PROGRAM C21_CamerasCtrl
VAR
END_VAR

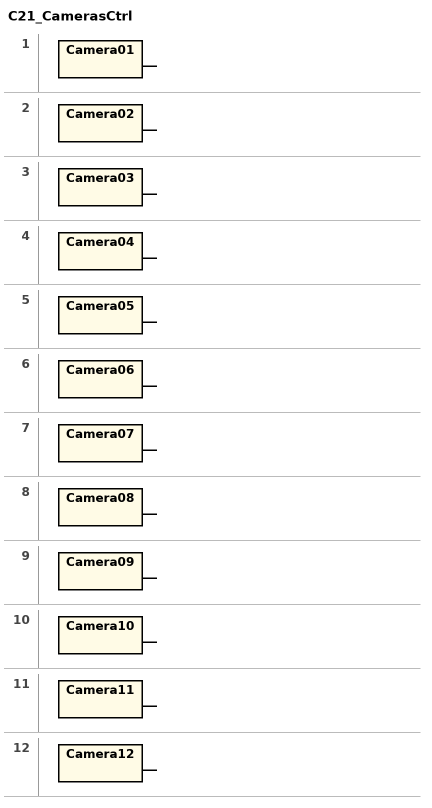
// NETWORK 1
Camera01();

// NETWORK 2
Camera02();

// NETWORK 3
Camera03();

// NETWORK 4
Camera04();

// NETWORK 5
Camera05();

// NETWORK 6
Camera06();

// NETWORK 7
Camera07();

// NETWORK 8
Camera08();

// NETWORK 9
Camera09();

// NETWORK 10
Camera10();

// NETWORK 11
Camera11();

// NETWORK 12
Camera12();

ACTION Camera01:
(*********************************************************CAMERA 01**********************************************************************)

(*stMasterListCameraOptions		: ST_SCANNER_Options := (eScannerType := E_MV_420_FULL, nImageBuffer := 1, nExpectedResp := 1);*)
IF gProcess.ePackAggregationMode <> E_SYSTEM_PAOL_2CAM AND gProcess.ePackAggregationMode <> E_SYSTEM_PAOL_3CAM  THEN

	gDevice.aCameraLightingIntensity[1] := F_SCANNER_LightingIntensity(gDevice.stMachineConfig.aCameraSettings[1].nLightingIntensity);

	gDevice.aCameraControl[1].stOptions.bUseExternalLight := gDevice.stMachineConfig.aCameraSettings[1].bUseExternalLight;
	gDevice.aCameraControl[1].stOptions.eScannerType	:= gDevice.stMachineConfig.aCameraSettings[1].eScannerType;

	IF gDevice.aCameraControl[1].stOptions.eScannerType = E_SCANNER_DeviceType.V430F THEN

		gDevice.aCameraControl[1].stOptions.nImageBuffer	:= 1;
		gDevice.aCameraControl[1].stOptions.nExpectedResp := 1;
		gDevice.aCameraControl[1].nReqProgram := 1;

	ELSE

		gDevice.aCameraControl[1].stOptions.nImageBuffer 	:= gDevice.stMachineConfig.aCameraSettings[1].nImageBuffer;
		gDevice.aCameraControl[1].stOptions.nExpectedResp := gDevice.stMachineConfig.aCameraSettings[1].nExpectedResp;

		CASE gDevice.stMachineConfig.aCameraSettings[1].eExpectedType OF
				E_SCANNER_CodeType.DATAMARTIX:
					gDevice.aCameraControl[1].nReqProgram := 1;
				E_SCANNER_CodeType.DOTCODE:
					gDevice.aCameraControl[1].nReqProgram := 2;
				E_SCANNER_CodeType.QR:
					gDevice.aCameraControl[1].nReqProgram := 3;
				E_SCANNER_CodeType.CODE128:
					gDevice.aCameraControl[1].nReqProgram := 4;
			ELSE
				gDevice.aCameraControl[1].nReqProgram := 1;
			END_CASE
	END_IF
END_IF
END_ACTION

ACTION Camera02:
(*********************************************************CAMERA 02**********************************************************************)
(*stPackAggregationCameraOptions		: ST_SCANNER_Options := (eScannerType := E_MV_420_FULL, nImageBuffer := 1, nExpectedResp := 1);*)
(*stPackAggregationCameraOptions		: ST_SCANNER_Options := (eScannerType := E_MV_None, nImageBuffer := 1, nExpectedResp := 5);*)
(*stPackAggregationCameraOptions		: ST_SCANNER_Options := (eScannerType := E_MV_None, nImageBuffer := 1, nExpectedResp := 2);*)
IF gProcess.ePackAggregationMode <> E_SYSTEM_PAOL_2CAM AND gProcess.ePackAggregationMode <> E_SYSTEM_PAOL_3CAM  THEN

	gDevice.aCameraLightingIntensity[2] := F_SCANNER_LightingIntensity(gDevice.stMachineConfig.aCameraSettings[2].nLightingIntensity);

	gDevice.aCameraControl[2].stOptions.bUseExternalLight := gDevice.stMachineConfig.aCameraSettings[2].bUseExternalLight;
	gDevice.aCameraControl[2].stOptions.eScannerType	:= gDevice.stMachineConfig.aCameraSettings[2].eScannerType;

	IF gDevice.aCameraControl[2].stOptions.eScannerType = E_SCANNER_DeviceType.V430F THEN

		gDevice.aCameraControl[2].stOptions.nImageBuffer	:= 1;
		gDevice.aCameraControl[2].stOptions.nExpectedResp := 1;
		gDevice.aCameraControl[2].nReqProgram := 1;

	ELSE

		gDevice.aCameraControl[2].stOptions.nImageBuffer 	:= gDevice.stMachineConfig.aCameraSettings[2].nImageBuffer;
		gDevice.aCameraControl[2].stOptions.nExpectedResp := gDevice.stMachineConfig.aCameraSettings[2].nExpectedResp;

		CASE gDevice.stMachineConfig.aCameraSettings[2].eExpectedType OF
				E_SCANNER_CodeType.DATAMARTIX:
					gDevice.aCameraControl[2].nReqProgram := 1;
				E_SCANNER_CodeType.DOTCODE:
					gDevice.aCameraControl[2].nReqProgram := 2;
				E_SCANNER_CodeType.QR:
					gDevice.aCameraControl[2].nReqProgram := 3;
				E_SCANNER_CodeType.CODE128:
					gDevice.aCameraControl[2].nReqProgram := 4;
			ELSE
				gDevice.aCameraControl[2].nReqProgram := 1;
			END_CASE
	END_IF
END_IF
END_ACTION

ACTION Camera03:
(*********************************************************CAMERA 03**********************************************************************)

(*stPackAggregationCameraOptions		: ST_SCANNER_Options := (eScannerType := E_MV_420_FULL, nImageBuffer := 1, nExpectedResp := 1);*)
(*stPackAggregationCameraOptions		: ST_SCANNER_Options := (eScannerType := E_MV_None, nImageBuffer := 1, nExpectedResp := 5);*)
(*stPackAggregationCameraOptions		: ST_SCANNER_Options := (eScannerType := E_MV_None, nImageBuffer := 1, nExpectedResp := 2);*)
IF gProcess.ePackAggregationMode <> E_SYSTEM_PAOL_2CAM AND gProcess.ePackAggregationMode <> E_SYSTEM_PAOL_3CAM  THEN

	gDevice.aCameraLightingIntensity[3] := F_SCANNER_LightingIntensity(gDevice.stMachineConfig.aCameraSettings[3].nLightingIntensity);

	gDevice.aCameraControl[3].stOptions.bUseExternalLight := gDevice.stMachineConfig.aCameraSettings[3].bUseExternalLight;
	gDevice.aCameraControl[3].stOptions.eScannerType	:= gDevice.stMachineConfig.aCameraSettings[3].eScannerType;

	IF gDevice.aCameraControl[3].stOptions.eScannerType = E_SCANNER_DeviceType.V430F THEN

		gDevice.aCameraControl[3].stOptions.nImageBuffer	:= 1;
		gDevice.aCameraControl[3].stOptions.nExpectedResp := 1;
		gDevice.aCameraControl[3].nReqProgram := 1;

	ELSE

		gDevice.aCameraControl[3].stOptions.nImageBuffer 	:= gDevice.stMachineConfig.aCameraSettings[3].nImageBuffer;
		gDevice.aCameraControl[3].stOptions.nExpectedResp := gDevice.stMachineConfig.aCameraSettings[3].nExpectedResp;

		CASE gDevice.stMachineConfig.aCameraSettings[3].eExpectedType OF
				E_SCANNER_CodeType.DATAMARTIX:
					gDevice.aCameraControl[3].nReqProgram := 1;
				E_SCANNER_CodeType.DOTCODE:
					gDevice.aCameraControl[3].nReqProgram := 2;
				E_SCANNER_CodeType.QR:
					gDevice.aCameraControl[3].nReqProgram := 3;
				E_SCANNER_CodeType.CODE128:
					gDevice.aCameraControl[3].nReqProgram := 4;
			ELSE
				gDevice.aCameraControl[3].nReqProgram := 1;
			END_CASE
	END_IF
END_IF
END_ACTION

ACTION Camera04:
(*********************************************************CAMERA 04**********************************************************************)
gDevice.aCameraLightingIntensity[4] := F_SCANNER_LightingIntensity(gDevice.stMachineConfig.aCameraSettings[4].nLightingIntensity);

gDevice.aCameraControl[4].stOptions.bUseExternalLight := gDevice.stMachineConfig.aCameraSettings[4].bUseExternalLight;
gDevice.aCameraControl[4].stOptions.eScannerType	:= gDevice.stMachineConfig.aCameraSettings[4].eScannerType;

IF gDevice.aCameraControl[4].stOptions.eScannerType = E_SCANNER_DeviceType.V430F THEN

	gDevice.aCameraControl[4].stOptions.nImageBuffer	:= 1;
	gDevice.aCameraControl[4].stOptions.nExpectedResp := 1;
	gDevice.aCameraControl[4].nReqProgram := 1;

ELSE

	gDevice.aCameraControl[4].stOptions.nImageBuffer 	:= gDevice.stMachineConfig.aCameraSettings[4].nImageBuffer;
	gDevice.aCameraControl[4].stOptions.nExpectedResp := gDevice.stMachineConfig.aCameraSettings[4].nExpectedResp;

	CASE gDevice.stMachineConfig.aCameraSettings[4].eExpectedType OF
			E_SCANNER_CodeType.DATAMARTIX:
				gDevice.aCameraControl[4].nReqProgram := 1;
			E_SCANNER_CodeType.DOTCODE:
				gDevice.aCameraControl[4].nReqProgram := 2;
			E_SCANNER_CodeType.QR:
				gDevice.aCameraControl[4].nReqProgram := 3;
			E_SCANNER_CodeType.CODE128:
				gDevice.aCameraControl[4].nReqProgram := 4;
		ELSE
			gDevice.aCameraControl[4].nReqProgram := 1;
		END_CASE
END_IF
END_ACTION

ACTION Camera05:
(*********************************************************CAMERA 05**********************************************************************)
gDevice.aCameraLightingIntensity[5] := F_SCANNER_LightingIntensity(gDevice.stMachineConfig.aCameraSettings[5].nLightingIntensity);

gDevice.aCameraControl[5].stOptions.bUseExternalLight := gDevice.stMachineConfig.aCameraSettings[5].bUseExternalLight;
gDevice.aCameraControl[5].stOptions.eScannerType	:= gDevice.stMachineConfig.aCameraSettings[5].eScannerType;
gDevice.aCameraControl[5].stOptions.nImageBuffer 	:= gDevice.stMachineConfig.aCameraSettings[5].nImageBuffer;
gDevice.aCameraControl[5].stOptions.nExpectedResp := gDevice.stMachineConfig.aCameraSettings[5].nExpectedResp;

CASE gDevice.stMachineConfig.aCameraSettings[5].eExpectedType OF
	E_SCANNER_CodeType.DATAMARTIX:
		gDevice.aCameraControl[5].nReqProgram := 1;
	E_SCANNER_CodeType.DOTCODE:
		gDevice.aCameraControl[5].nReqProgram := 2;
	E_SCANNER_CodeType.QR:
		gDevice.aCameraControl[5].nReqProgram := 3;
	E_SCANNER_CodeType.CODE128:
		gDevice.aCameraControl[5].nReqProgram := 4;
ELSE
	gDevice.aCameraControl[5].nReqProgram := 1;
END_CASE
END_ACTION

ACTION Camera06:
(*********************************************************CAMERA 06**********************************************************************)
gDevice.aCameraLightingIntensity[6] := F_SCANNER_LightingIntensity(gDevice.stMachineConfig.aCameraSettings[6].nLightingIntensity);

gDevice.aCameraControl[6].stOptions.bUseExternalLight := gDevice.stMachineConfig.aCameraSettings[6].bUseExternalLight;
gDevice.aCameraControl[6].stOptions.eScannerType	:= gDevice.stMachineConfig.aCameraSettings[6].eScannerType;
gDevice.aCameraControl[6].stOptions.nImageBuffer 	:= gDevice.stMachineConfig.aCameraSettings[6].nImageBuffer;
gDevice.aCameraControl[6].stOptions.nExpectedResp := gDevice.stMachineConfig.aCameraSettings[6].nExpectedResp;

CASE gDevice.stMachineConfig.aCameraSettings[6].eExpectedType OF
	E_SCANNER_CodeType.DATAMARTIX:
		gDevice.aCameraControl[6].nReqProgram := 1;
	E_SCANNER_CodeType.DOTCODE:
		gDevice.aCameraControl[6].nReqProgram := 2;
	E_SCANNER_CodeType.QR:
		gDevice.aCameraControl[6].nReqProgram := 3;
	E_SCANNER_CodeType.CODE128:
		gDevice.aCameraControl[6].nReqProgram := 4;
ELSE
	gDevice.aCameraControl[6].nReqProgram := 1;
END_CASE
END_ACTION

ACTION Camera07:
(*********************************************************CAMERA 07**********************************************************************)
gDevice.aCameraLightingIntensity[7] := F_SCANNER_LightingIntensity(gDevice.stMachineConfig.aCameraSettings[7].nLightingIntensity);

gDevice.aCameraControl[7].stOptions.bUseExternalLight := gDevice.stMachineConfig.aCameraSettings[7].bUseExternalLight;
gDevice.aCameraControl[7].stOptions.eScannerType	:= gDevice.stMachineConfig.aCameraSettings[7].eScannerType;

IF gDevice.aCameraControl[7].stOptions.eScannerType = E_SCANNER_DeviceType.V430F THEN

	gDevice.aCameraControl[7].stOptions.nImageBuffer	:= 1;
	gDevice.aCameraControl[7].stOptions.nExpectedResp := 1;
	gDevice.aCameraControl[7].nReqProgram := 1;

ELSE

	gDevice.aCameraControl[7].stOptions.nImageBuffer 	:= gDevice.stMachineConfig.aCameraSettings[7].nImageBuffer;

	IF gDevice.stMachineConfig.bMasterListCameraDoubleRead AND NOT gDevice.stMachineConfig.bEANValidationEnable THEN
		gDevice.aCameraControl[7].stOptions.nExpectedResp := 2;
	ELSE
		gDevice.aCameraControl[7].stOptions.nExpectedResp := gDevice.stMachineConfig.aCameraSettings[7].nExpectedResp;
	END_IF

	CASE gDevice.stMachineConfig.aCameraSettings[7].eExpectedType OF
			E_SCANNER_CodeType.DATAMARTIX:
				gDevice.aCameraControl[7].nReqProgram := 1;
			E_SCANNER_CodeType.DOTCODE:
				gDevice.aCameraControl[7].nReqProgram := 2;
			E_SCANNER_CodeType.QR:
				gDevice.aCameraControl[7].nReqProgram := 3;
			E_SCANNER_CodeType.CODE128:
				gDevice.aCameraControl[7].nReqProgram := 4;
		ELSE
			gDevice.aCameraControl[7].nReqProgram := 1;
		END_CASE
END_IF
END_ACTION

ACTION Camera08:
(*********************************************************CAMERA 08**********************************************************************)
gDevice.aCameraLightingIntensity[8] := F_SCANNER_LightingIntensity(gDevice.stMachineConfig.aCameraSettings[8].nLightingIntensity);

gDevice.aCameraControl[8].stOptions.bUseExternalLight := gDevice.stMachineConfig.aCameraSettings[8].bUseExternalLight;
gDevice.aCameraControl[8].stOptions.eScannerType	:= gDevice.stMachineConfig.aCameraSettings[8].eScannerType;

IF gDevice.aCameraControl[8].stOptions.eScannerType = E_SCANNER_DeviceType.V430F THEN

	gDevice.aCameraControl[8].stOptions.nImageBuffer	:= 1;
	gDevice.aCameraControl[8].stOptions.nExpectedResp := 1;
	gDevice.aCameraControl[8].nReqProgram := 1;

ELSE

	gDevice.aCameraControl[8].stOptions.nImageBuffer 	:= gDevice.stMachineConfig.aCameraSettings[8].nImageBuffer;
	gDevice.aCameraControl[8].stOptions.nExpectedResp := gDevice.stMachineConfig.aCameraSettings[8].nExpectedResp;


	IF gDevice.aCameraControl[8].stOptions.nExpectedResp = 2 THEN

		CASE gDevice.stMachineConfig.aCameraSettings[8].eExpectedType OF
			E_SCANNER_CodeType.DATAMARTIX:
				gDevice.aCameraControl[8].nReqProgram := 2;
			E_SCANNER_CodeType.DOTCODE:
				gDevice.aCameraControl[8].nReqProgram := 4;
			E_SCANNER_CodeType.QR:
				gDevice.aCameraControl[8].nReqProgram := 6;
			E_SCANNER_CodeType.CODE128:
				gDevice.aCameraControl[8].nReqProgram := 8;
		ELSE
			gDevice.aCameraControl[8].nReqProgram := 2;
		END_CASE
	ELSE
		CASE gDevice.stMachineConfig.aCameraSettings[8].eExpectedType OF
			E_SCANNER_CodeType.DATAMARTIX:
				gDevice.aCameraControl[8].nReqProgram := 1;
			E_SCANNER_CodeType.DOTCODE:
				gDevice.aCameraControl[8].nReqProgram := 3;
			E_SCANNER_CodeType.QR:
				gDevice.aCameraControl[8].nReqProgram := 5;
			E_SCANNER_CodeType.CODE128:
				gDevice.aCameraControl[8].nReqProgram := 7;
		ELSE
			gDevice.aCameraControl[8].nReqProgram := 1;
		END_CASE
	END_IF

END_IF
END_ACTION

ACTION Camera09:
(*********************************************************CAMERA 09**********************************************************************)
gDevice.aCameraLightingIntensity[9] := F_SCANNER_LightingIntensity(gDevice.stMachineConfig.aCameraSettings[9].nLightingIntensity);

gDevice.aCameraControl[9].stOptions.bUseExternalLight := gDevice.stMachineConfig.aCameraSettings[9].bUseExternalLight;
gDevice.aCameraControl[9].stOptions.eScannerType	:= gDevice.stMachineConfig.aCameraSettings[9].eScannerType;

IF gDevice.aCameraControl[9].stOptions.eScannerType = E_SCANNER_DeviceType.V430F THEN

	gDevice.aCameraControl[9].stOptions.nImageBuffer	:= 1;
	gDevice.aCameraControl[9].stOptions.nExpectedResp := 1;
	gDevice.aCameraControl[9].nReqProgram := 1;

ELSIF gDevice.stMachineConfig.bPassthrough AND gDevice.stMachineConfig.bEANValidationEnable THEN

	gDevice.aCameraControl[9].stOptions.nImageBuffer	:= 1;
	gDevice.aCameraControl[9].stOptions.nExpectedResp := 1;
	gDevice.aCameraControl[9].nReqProgram := 3;

ELSE

	gDevice.aCameraControl[9].stOptions.nImageBuffer 	:= gDevice.stMachineConfig.aCameraSettings[9].nImageBuffer;

	IF gDevice.stMachineConfig.bMasterListCameraDoubleRead  THEN

		gDevice.aCameraControl[9].stOptions.nExpectedResp := 2;
	ELSE
		gDevice.aCameraControl[9].stOptions.nExpectedResp := gDevice.stMachineConfig.aCameraSettings[9].nExpectedResp;
	END_IF

	IF gDevice.aCameraControl[9].stOptions.nExpectedResp = 2 THEN

		CASE gDevice.stMachineConfig.aCameraSettings[9].eExpectedType OF
			E_SCANNER_CodeType.DATAMARTIX:
				gDevice.aCameraControl[9].nReqProgram := 2;
			E_SCANNER_CodeType.DOTCODE:
				gDevice.aCameraControl[9].nReqProgram := 4;
			E_SCANNER_CodeType.QR:
				gDevice.aCameraControl[9].nReqProgram := 6;
			E_SCANNER_CodeType.CODE128:
				gDevice.aCameraControl[9].nReqProgram := 8;
		ELSE
			gDevice.aCameraControl[9].nReqProgram := 2;
		END_CASE
	ELSE
		CASE gDevice.stMachineConfig.aCameraSettings[9].eExpectedType OF
			E_SCANNER_CodeType.DATAMARTIX:
				gDevice.aCameraControl[9].nReqProgram := 1;
			E_SCANNER_CodeType.DOTCODE:
				gDevice.aCameraControl[9].nReqProgram := 3;
			E_SCANNER_CodeType.QR:
				gDevice.aCameraControl[9].nReqProgram := 5;
			E_SCANNER_CodeType.CODE128:
				gDevice.aCameraControl[9].nReqProgram := 7;
		ELSE
			gDevice.aCameraControl[9].nReqProgram := 1;
		END_CASE
	END_IF
END_IF
END_ACTION

ACTION Camera10:
(*********************************************************CAMERA 10**********************************************************************)
gDevice.aCameraLightingIntensity[10] := F_SCANNER_LightingIntensity(gDevice.stMachineConfig.aCameraSettings[10].nLightingIntensity);

gDevice.aCameraControl[10].stOptions.bUseExternalLight := gDevice.stMachineConfig.aCameraSettings[10].bUseExternalLight;
gDevice.aCameraControl[10].stOptions.eScannerType	:= gDevice.stMachineConfig.aCameraSettings[10].eScannerType;

IF gDevice.aCameraControl[10].stOptions.eScannerType = E_SCANNER_DeviceType.V430F THEN

	gDevice.aCameraControl[10].stOptions.nImageBuffer	:= 1;
	gDevice.aCameraControl[10].stOptions.nExpectedResp := 1;
	gDevice.aCameraControl[10].nReqProgram := 1;

ELSE

	gDevice.aCameraControl[10].stOptions.nImageBuffer 	:= gDevice.stMachineConfig.aCameraSettings[10].nImageBuffer;
	gDevice.aCameraControl[10].stOptions.nExpectedResp := gDevice.stMachineConfig.aCameraSettings[10].nExpectedResp;

	CASE gDevice.stMachineConfig.aCameraSettings[10].eExpectedType OF
			E_SCANNER_CodeType.DATAMARTIX:
				gDevice.aCameraControl[10].nReqProgram := 1;
			E_SCANNER_CodeType.DOTCODE:
				gDevice.aCameraControl[10].nReqProgram := 2;
			E_SCANNER_CodeType.QR:
				gDevice.aCameraControl[10].nReqProgram := 3;
			E_SCANNER_CodeType.CODE128:
				gDevice.aCameraControl[10].nReqProgram := 4;
		ELSE
			gDevice.aCameraControl[10].nReqProgram := 1;
		END_CASE
END_IF
END_ACTION

ACTION Camera11:
(*********************************************************CAMERA 11**********************************************************************)
gDevice.aCameraLightingIntensity[11] := F_SCANNER_LightingIntensity(gDevice.stMachineConfig.aCameraSettings[11].nLightingIntensity);

gDevice.aCameraControl[11].stOptions.bUseExternalLight := gDevice.stMachineConfig.aCameraSettings[11].bUseExternalLight;
gDevice.aCameraControl[11].stOptions.eScannerType	:= gDevice.stMachineConfig.aCameraSettings[11].eScannerType;

IF gDevice.aCameraControl[11].stOptions.eScannerType = E_SCANNER_DeviceType.V430F THEN

	gDevice.aCameraControl[11].stOptions.nImageBuffer	:= 1;
	gDevice.aCameraControl[11].stOptions.nExpectedResp := 1;
	gDevice.aCameraControl[11].nReqProgram := 1;

ELSE

	gDevice.aCameraControl[11].stOptions.nImageBuffer 	:= gDevice.stMachineConfig.aCameraSettings[11].nImageBuffer;
	gDevice.aCameraControl[11].stOptions.nExpectedResp := gDevice.stMachineConfig.aCameraSettings[11].nExpectedResp;

	CASE gDevice.stMachineConfig.aCameraSettings[11].eExpectedType OF
			E_SCANNER_CodeType.DATAMARTIX:
				gDevice.aCameraControl[11].nReqProgram := 1;
			E_SCANNER_CodeType.DOTCODE:
				gDevice.aCameraControl[11].nReqProgram := 2;
			E_SCANNER_CodeType.QR:
				gDevice.aCameraControl[11].nReqProgram := 3;
			E_SCANNER_CodeType.CODE128:
				gDevice.aCameraControl[11].nReqProgram := 4;
		ELSE
			gDevice.aCameraControl[11].nReqProgram := 1;
		END_CASE
END_IF
END_ACTION

ACTION Camera12:
(*********************************************************CAMERA 12**********************************************************************)
gDevice.aCameraLightingIntensity[12] := F_SCANNER_LightingIntensity(gDevice.stMachineConfig.aCameraSettings[12].nLightingIntensity);

gDevice.aCameraControl[12].stOptions.bUseExternalLight := gDevice.stMachineConfig.aCameraSettings[12].bUseExternalLight;
gDevice.aCameraControl[12].stOptions.eScannerType	:= gDevice.stMachineConfig.aCameraSettings[12].eScannerType;

IF gDevice.aCameraControl[12].stOptions.eScannerType = E_SCANNER_DeviceType.V430F THEN

	gDevice.aCameraControl[12].stOptions.nImageBuffer	:= 1;
	gDevice.aCameraControl[12].stOptions.nExpectedResp := 1;
	gDevice.aCameraControl[12].nReqProgram := 1;

ELSIF gDevice.stMetsStatus.stPCMStatus.nOpMode < 7 THEN

	gDevice.aCameraControl[12].stOptions.nImageBuffer	:= 1;
	gDevice.aCameraControl[12].stOptions.nExpectedResp := 1;
	gDevice.aCameraControl[12].nReqProgram := 5;

ELSE

	gDevice.aCameraControl[12].stOptions.nImageBuffer 	:= gDevice.stMachineConfig.aCameraSettings[12].nImageBuffer;
	gDevice.aCameraControl[12].stOptions.nExpectedResp := gDevice.stMachineConfig.aCameraSettings[12].nExpectedResp;

	CASE gDevice.stMachineConfig.aCameraSettings[12].eExpectedType OF
			E_SCANNER_CodeType.DATAMARTIX:
				gDevice.aCameraControl[12].nReqProgram := 1;
			E_SCANNER_CodeType.DOTCODE:
				gDevice.aCameraControl[12].nReqProgram := 2;
			E_SCANNER_CodeType.QR:
				gDevice.aCameraControl[12].nReqProgram := 3;
			E_SCANNER_CodeType.CODE128:
				gDevice.aCameraControl[12].nReqProgram := 4;
		ELSE
			gDevice.aCameraControl[12].nReqProgram := 1;
		END_CASE
END_IF
END_ACTION

END_PROGRAM

(* stored: Version 1.1.0.1
   POU C21_CamerasCtrl: Id {2037e324-dea3-4f0c-806a-b675c4c0e95a}, SpecialFunc None
   Action Camera01: Id {d9410514-f5a0-4cd7-b192-96147cc84076}
   Action Camera02: Id {fd089a61-2748-49c3-a78a-a8f7930551e9}
   Action Camera03: Id {0c24c973-69ad-4e38-92d4-2e815ec5051a}
   Action Camera04: Id {118670b7-c542-4a0f-bed4-00506a5fe966}
   Action Camera05: Id {10ef1c76-670b-44ec-b902-44a38a23e7c9}
   Action Camera06: Id {398d5066-34a1-413d-9ce8-a0e0bc0a9858}
   Action Camera07: Id {56f527e9-b6be-4c6a-a391-2ba6e4e1fc6a}
   Action Camera08: Id {0f55681b-10b9-4a23-baf9-625b1e8f9e5d}
   Action Camera09: Id {c7ae0c68-2f49-4b23-b98f-0d9ac65534a8}
   Action Camera10: Id {b3181e0d-72ba-46e6-8516-701bfaec35a0}
   Action Camera11: Id {0f8b38eb-1911-4d68-aabf-cc764ae63cbf}
   Action Camera12: Id {ecfccefb-3927-4f0c-9372-3a1ca5f9b0d8} *)
